{attribute 'qualified_only'}
{attribute 'strict'}
TYPE E_StewartOpMode :
(
	MANUAL := 16#00,
	NORMAL := 16#01
) USINT;
END_TYPE

(* stored: Version 1.1.0.1, ProductVersion 3.1.4022.18
   DUT E_StewartOpMode: Id {063aec99-d750-4f47-b1e1-153470d88024} *)
